PROGRAM MAIN
VAR
END_VAR

//This is my

END_PROGRAM

(* stored: Version 1.1.0.1, ProductVersion 3.1.4024.4
   POU MAIN: Id {c02bc9fe-10ce-49e8-a335-4a980b9491e9}, SpecialFunc None *)
